// TIA Portal V20 export
// export: Created 2026-09-14T11:29:27.957232Z, ExportSetting None, DisplayName Totally Integrated Automation Portal, DisplayVersion V20, DisplayName TIA Portal Openness, DisplayVersion V20, DisplayName TIA Portal Version Control Interface, DisplayVersion V20, DisplayName STEP 7 Professional, DisplayVersion V20, DisplayName STEP 7 Safety, DisplayVersion V20, DisplayName WinCC Basic/Comfort/Advanced, DisplayVersion V20, DisplayName WinCC Unified, DisplayVersion V20
VAR_GLOBAL   // PLC tag table "Sorting Plant Tags"
   csLightSensorCube_Detected AT %I0.0 : Bool;   // 0: cube workpiece not detected; 1: cube workpiece detected by the light sensor
   csLightSensorCylinder_Detected AT %I0.1 : Bool;   // 0: cylinder workpiece not detected; 1: cylinder workpiece detected by the light sensor
   csLightSensorWorkpiece_Detected AT %I0.2 : Bool;   // 0: light sensor did not detect a workpiece, 1: light sensor detected a workpiece
   csLimitSwitchCylinderNotExtended_Activated AT %I0.3 : Bool;   // 0: the cylinder is fully extended; 1: the cylinder is not fully extended
   csLimitSwitchCylinderRetracted_Activated AT %I0.4 : Bool;   // 0: the cylinder is not fully retracted; 1: the cylinder is fully retracted
   osWorkpieceCylinder_SetActive AT %Q0.0 : Bool;   // 0: cylinder workpiece are not produced; 1: cylinder workpiece are produced
   osWorkpieceCube_SetActive AT %Q0.1 : Bool;   // 0: cube workpiece are not produced; 1: cube workpiece are produced
   pcCylinderHeadRetract_SetActive AT %Q0.2 : Bool;   // 0: do not retract push cylinder; 1: retract push cylinder
   pcCylinderHeadExtend_SetActive AT %Q0.3 : Bool;   // 0: do not extend push cylinder; 1: extend push cylinder
   scConveyorLongConstSpeed_SetActive AT %Q0.4 : Bool;   // 0: do not move the long conveyor at constant speed; 1: move the long conveyor at constant speed
   scConveyorLongVarSpeed_SetActive AT %Q0.5 : Bool;   // 0: do not move the long conveyor at variable speed; 1: move the long conveyor at variable speed
   scConveyorShortConstSpeed_SetActive AT %Q0.6 : Bool;   // 0: do not move the short conveyor at constant speed; 1: move the short conveyor at constant speed
   scConveyorShortVarSpeed_SetActive AT %Q0.7 : Bool;   // 0: do not move the short conveyor at variable speed; 1: move the short conveyor at variable speed
   scConveyorLongVarSpeed_SetSpeed AT %QD64 : Real;   // variable velocity for long conveyor belt in m/s
   scConveyorShortVarSpeed_SetSpeed AT %QD68 : Real;   // variable velocity for short conveyor belt in m/s
END_VAR
